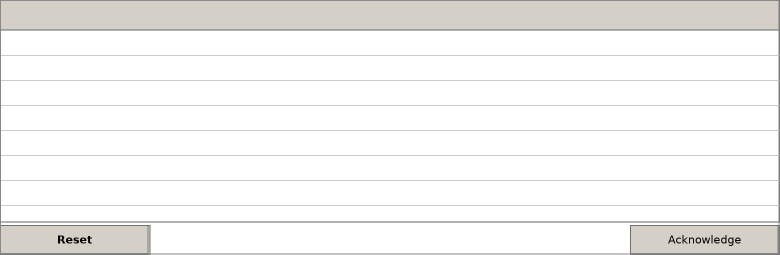
VISUALIZATION LogView  // 780x255
VAR_IN_OUT
	arLog : ARRAY[1..10] OF UDT_LogItem; // Array size must match declaration in FB_LogView!
	bAcknowledge : BOOL; // Clear inactive faults from the log
	bReset : BOOL; // Triggers a reset 
END_VAR
    Table (0,0 780x222), data array: arLog
        p3854506369: arLog[INDEX].Id
        p1892666644: arLog[INDEX].sID
        p338671338: arLog[INDEX].sDescription
        p2170511999: arLog[INDEX].sStartTime
        p3723444502: arLog[INDEX].sEndTime
        p2232123230: arLog[INDEX].bAlarmState
        Columns.Column.[0].Template: arLog[INDEX].stFault.Active
    Button (630,225 150x30), "Acknowledge"
        tap bAcknowledge
    Button (0,225 150x30), "Reset"
        tap bReset
END_VISUALIZATION

(* stored: Version 1.1.0.1, ProductVersion 3.1.4024.11
   Visu LogView: Id {07ec0c4a-ff40-487e-8918-11af5123365d} *)
